FUNCTION_BLOCK PUBLIC EventLogger
VAR_INPUT
	eEventType : E_eventType ;
	nEventIdentity : UDINT ;
	strEventText	: STRING(255);
END_VAR

VAR
	EventBuffer : ARRAY [1..Max_Size_OF_Buffer] OF ST_Event;
	CurrentEventBufferIndex : INT:= 0;
	i 						: INT;
END_VAR

VAR CONSTANT
	Max_Size_OF_Buffer : INT := 100;
END_VAR

FOR i :=  Max_Size_OF_Buffer TO 2 BY -1 DO 
	EventBuffer[i]:= EventBuffer[i-1];
END_FOR
EventBuffer[1].eEventType := eEventType;
EventBuffer[1].nEventIdentity	:= nEventIdentity;
EventBuffer[1].strEventText	:= strEventText;
UpdateEventTimeWithSystemTime(stEvent := EventBuffer[1]);

END_FUNCTION_BLOCK

(* stored: Version 1.1.0.1, ProductVersion 3.1.4024.15
   POU EventLogger: Id {1aba1ebd-9bd9-47c4-9870-a817908ee061}, SpecialFunc None *)
